(* IEC 61131-3 sources: CSVCore/src/Ar/CSVCore, 3 files *)

(* ---- Types.typ ---- *)
(*
 * File: Types.typ
 * Copyright (c) 2023 Loupe
 * https://loupe.team
 *
 * This file is part of CSVCore, licensed under the MIT License.
 *
 *)

TYPE
	CSVCoreCfg_typ : 	STRUCT
		delim : USINT := 44; (*Delimiter seperating cells. Defualt ','*)
		comment : STRING[5] := '//'; (*Characters representing line comments*)
		headerRow : UDINT := 0; (*Row number containing header. 0 means no header*)
		quoteCharacter : USINT := 34; (*Quote character to be used for building csv data. Defualt "*)
		quoteUnescaping : {REDUND_UNREPLICABLE} BOOL := TRUE; (*Unescape quoted strings*)
		forceEscaping : BOOL := FALSE; (*Force strings to be escaped when building csv data*)
		ignoreEmptyRows : BOOL := TRUE; (*Skip Rows that have no values. Not fully implemented*)
	END_STRUCT;
	CSVCoreOut_typ : 	STRUCT
		headerRow : UDINT;
		rowNumber : UDINT;
		pRow : UDINT;
		rowLen : UDINT;
	END_STRUCT;
	CSVCore_typ : 	STRUCT
		predef : CSVPredef_typ;
		cfg : CSVCoreCfg_typ;
		out : CSVCoreOut_typ;
		internal : CSVCoreInternal_typ;
	END_STRUCT;
	CSVCoreInternal_typ : 	STRUCT
		rowNumber : DINT;
		pRow : UDINT;
		rowLen : UDINT;
		pData : UDINT;
		dataSize : UDINT;
	END_STRUCT;
	CSVPredef_typ : 	STRUCT
		numColumns : USINT;
		pColumns : UDINT;
		pTypes : UDINT;
		pStatus : UDINT;
	END_STRUCT;
	CSV_CORE_ERR_enum :
		(
		CSV_CORE_ERR_OK := 0,
		CSV_CORE_ERR_NO_NEWLINE := 5000,
		CSV_CORE_ERR_NEWLINE,
		CSV_CORE_ERR_END_OF_LINE,
		CSV_CORE_ERR_END_OF_DATA,
		CSV_CORE_ERR_BUFFER_FULL,
		CSV_CORE_ERR_HEADER_INDEX,
		CSV_CORE_ERR_NUM_COLUMNS,
		CSV_CORE_ERR_INVALID_INPUT,
		CSV_CORE_ERR_INTERNAL,
		CSV_CORE_ERR_COLUMN_NOT_FOUND,
		CSV_CORE_ERR_INVALID_VALUE,
		CSV_CORE_ERR_INVALID_TYPE,
		CSV_CORE_ERR_UNSUPPORTED_TYPE,
		CSV_CORE_ERR_NOT_IMPLEMENTED
		);
	CSV_CORE_TYPE_enum :
		(
		CSV_CORE_TYPE_STRUCT := 0, (*0*)
		CSV_CORE_TYPE_BOOL,
		CSV_CORE_TYPE_SINT,
		CSV_CORE_TYPE_INT,
		CSV_CORE_TYPE_DINT,
		CSV_CORE_TYPE_USINT, (*5*)
		CSV_CORE_TYPE_UINT,
		CSV_CORE_TYPE_UDINT,
		CSV_CORE_TYPE_REAL,
		CSV_CORE_TYPE_STRING,
		CSV_CORE_TYPE_ULINT, (*10*)
		CSV_CORE_TYPE_DATE_AND_TIME,
		CSV_CORE_TYPE_TIME,
		CSV_CORE_TYPE_DATE,
		CSV_CORE_TYPE_LREAL,
		CSV_CORE_TYPE_ARRAY_OF_STRUCT, (*15*)
		CSV_CORE_TYPE_TIME_OF_DAY,
		CSV_CORE_TYPE_BYTE,
		CSV_CORE_TYPE_WORD,
		CSV_CORE_TYPE_DWORD,
		CSV_CORE_TYPE_LWORD, (*20*)
		CSV_CORE_TYPE_WSTRING, (*21*)
		CSV_CORE_TYPE_LINT := 23, (*23*)
		CSV_CORE_TYPE_STRINGN := 1000 (*1000*)
		);
END_TYPE

(* ---- CSVCore.fun ---- *)
(*
 * File: CSVCore.fun
 * Copyright (c) 2023 Loupe
 * https://loupe.team
 *
 * This file is part of CSVCore, licensed under the MIT License.
 *
 *)

(*Predef*)

FUNCTION csvInitPredef : DINT (*Initializes a Predef*)
	VAR_INPUT
		pPredef : CSVPredef_typ; (*Pointer to predef to initialize*)
		numColumns : UDINT; (*Number of columns Predef will return*)
		pColumns : UDINT; (*Pointer to array of INT size numColumns (optional)*)
		pTypes : UDINT; (*Pointer to array of CSV_CORE_TYPE_enum size numColumns (optional)*)
		pStatus : UDINT; (*Pointer to array of CSV_CORE_ERR_enum size numColumns (optional)*)
	END_VAR
END_FUNCTION

FUNCTION csvFilterByHeader : DINT (*Apply a filter by header to Predef*)
	VAR_INPUT
		pCsv : REFERENCE TO CSVCore_typ; (*Pointer to csv object containing data*)
		pPredef : CSVPredef_typ; (*Pointer to predef to apply filter to *)
		varArgs : UDINT; (*Optional number of arguments*)
	END_VAR
END_FUNCTION

FUNCTION csvFilterByColumn : DINT (*Apply a filter by columns to Predef*)
	VAR_INPUT
		pPredef : CSVPredef_typ; (*Pointer to predef to apply filter to*)
		varArgs : UDINT; (*Optional number of arguments*)
	END_VAR
END_FUNCTION

FUNCTION csvCastAs : DINT (*Apply types definitions to columnns in Predef*)
	VAR_INPUT
		pPredef : CSVPredef_typ; (*Pointer to predef to apply filter to *)
		varArgs : UDINT; (*Optional number of arguments*)
	END_VAR
END_FUNCTION

FUNCTION csvCastAllAs : DINT (*Apply type definition to all calomns in Predef*)
	VAR_INPUT
		pPredef : CSVPredef_typ; (*Pointer to predef to apply filter to *)
		dataType : CSV_CORE_TYPE_enum; (*Data type that columns should be formatted as*)
	END_VAR
END_FUNCTION

FUNCTION csvSetPredef : DINT (*Set defualt Predef*)
	VAR_INPUT
		pCsv : CSVCore_typ; (*Pointer to csv object*)
		pPredef : CSVPredef_typ; (*Pointer to predef to copy configuration from*)
	END_VAR
END_FUNCTION
(*Parsing*)

FUNCTION csvInitData : DINT (*Initialize csv object*)
	VAR_INPUT
		pCsv : CSVCore_typ; (*Pointer to csv object*)
		pData : UDINT; (*Pointer to container to contain csv data*)
		dataSize : UDINT; (*Size of data container*)
	END_VAR
END_FUNCTION

FUNCTION csvReadNextRow : DINT (*Read next row using default Predef*)
	VAR_INPUT
		pCsv : CSVCore_typ; (*Pointer to csv object*)
		varargs : UDINT; (*Optional number of arguments*)
	END_VAR
END_FUNCTION

FUNCTION csvReadRowAs : DINT (*ReRead row using Predef*)
	VAR_INPUT
		pCsv : CSVCore_typ; (*Pointer to csv object*)
		pPredef : CSVPredef_typ; (*Pointer to predef to use while parsing row*)
		varargs : UDINT; (*Optional number of arguments*)
	END_VAR
END_FUNCTION

FUNCTION csvReadNextRowAs : DINT
	VAR_INPUT
		pCsv : CSVCore_typ; (*Pointer to csv object*)
		pPredef : CSVPredef_typ; (*Pointer to predef to use while parsing row*)
		varargs : UDINT; (*Optional number of arguments*)
	END_VAR
END_FUNCTION
(*Building*)

FUNCTION csvBuildRow : DINT (*Build row and append to data*)
	VAR_INPUT
		pCsv : CSVCore_typ; (*Pointer to csv object*)
		varArgs : UDINT; (*Optional number of arguments*)
	END_VAR
END_FUNCTION

FUNCTION csvBuildRowAs : DINT (*Build row from predef and append to data*)
	VAR_INPUT
		pCsv : CSVCore_typ; (*Pointer to csv object*)
		pPredef : CSVPredef_typ; (*Pointer to predef to use while building row*)
		varArgs : UDINT; (*Optional number of arguments*)
	END_VAR
END_FUNCTION

FUNCTION csvBuildComment : DINT (*Build comment and append to data*)
	VAR_INPUT
		pCsv : CSVCore_typ; (*Pointer to csv object*)
		pComment : UDINT; (*Pointer to string containg comment to be appeneded*)
	END_VAR
END_FUNCTION

FUNCTION csvBuildCell : DINT (*Build cell and append to data*)
	VAR_INPUT
		pCsv : CSVCore_typ; (*Pointer to csv object*)
		pVar : UDINT; (*Pointer to variable containing data to be added row*)
		pType : CSV_CORE_TYPE_enum; (*Type of pVar*)
		appendEndOfLine : BOOL; (*Apply newline after cell*)
	END_VAR
END_FUNCTION

FUNCTION csvAppendRow : DINT (*Append row to data*)
	VAR_INPUT
		pCsv : CSVCore_typ; (*Pointer to csv object*)
		pRow : UDINT; (*Pointer to string containing row data*)
	END_VAR
END_FUNCTION
(*Advanced*)

FUNCTION csvGetLineLenFn : DINT (*get length of line*)
	VAR_INPUT
		pString : UDINT; (*Pointer to string*)
		pLen : UDINT; (*Pointer to UDINT to be populated with length*)
	END_VAR
END_FUNCTION

FUNCTION csvGetNextLineFn : DINT (*get next line*)
	VAR_INPUT
		ppString : UDINT; (*Pointer to Pointer to string. Pointer will be moved to start of next line*)
		pLen : UDINT; (*Pointer to UDINT to be populated with length (optional)*)
		skipEmptyLines : BOOL; (*Skip lines that contain no data*)
	END_VAR
END_FUNCTION

FUNCTION csvGetNLineFn : DINT (*get nth line*)
	VAR_INPUT
		ppString : UDINT; (*Pointer to Pointer to string. Pointer will be moved to start of next line*)
		pLen : UDINT; (*Pointer to UDINT to be populated with length (optional)*)
		lineNum : DINT; (*Zero indexed line number to get*)
		skipEmptyLines : BOOL; (*Skip lines that contain no data*)
	END_VAR
END_FUNCTION

FUNCTION csvGetCellLenFn : DINT (*get length of cell*)
	VAR_INPUT
		pString : UDINT; (*Pointer to string*)
		pLen : UDINT; (*Pointer to UDINT to be populated with length*)
		delim : USINT; (*Deliminator seperating cells*)
	END_VAR
END_FUNCTION

FUNCTION csvGetNextCellFn : DINT (*get next cell*)
	VAR_INPUT
		ppString : UDINT; (*Pointer to Pointer to string. Pointer will be moved to start of next cell*)
		pLen : UDINT; (*Pointer to UDINT to be populated with length (optional)*)
		delim : USINT; (*Deliminator seperating cells*)
	END_VAR
END_FUNCTION

FUNCTION csvGetNCellFn : DINT (*get nth cell*)
	VAR_INPUT
		ppString : UDINT; (*Pointer to Pointer to string. Pointer will be moved to start of next cell*)
		pLen : UDINT; (*Pointer to UDINT to be populated with length (optional)*)
		cellNum : DINT; (*Zero indexed cell number to get*)
		delim : USINT; (*Deliminator seperating cells*)
	END_VAR
END_FUNCTION

(* ---- Constants.var ---- *)
(*
 * File: Constants.var
 * Copyright (c) 2023 Loupe
 * https://loupe.team
 *
 * This file is part of CSVCore, licensed under the MIT License.
 *
 *)

VAR CONSTANT
	CSV_CORE_DEF_MAX_COLUMNS : USINT := 10;
	CSV_CORE_DEF_MAI_COLUMNS : USINT := CSV_CORE_DEF_MAX_COLUMNS-1;
	CSV_CORE_MAX_CHAR_REP : UINT := 65;
END_VAR
(*Data type limits*)
VAR CONSTANT
	CSV_CORE_MIN_SINT : DINT := -128;
	CSV_CORE_MAX_SINT : DINT := 127;
	CSV_CORE_MIN_INT : DINT := -32768;
	CSV_CORE_MAX_INT : DINT := 32767;
	CSV_CORE_MIN_DINT : DINT := -2147483647;
	CSV_CORE_MAX_DINT : DINT := 2147483647;
	CSV_CORE_MIN_USINT : DINT := 0;
	CSV_CORE_MAX_USINT : DINT := 255;
	CSV_CORE_MIN_UINT : DINT := 0;
	CSV_CORE_MAX_UINT : DINT := 65535;
	CSV_CORE_MIN_UDINT : UDINT := 0;
	CSV_CORE_MAX_UDINT : UDINT := 4294967295;
	CSV_CORE_MIN_REAL : REAL := -3.4E038;
	CSV_CORE_MAX_REAL : REAL := 3.4E038;
END_VAR
